(* CODESYS project GVL_CELL_MANAGER.gvl.xml

Project tree, tasks and I/O mapping:
  global variables GVL_CELL_MANAGER
*)

// GVL_CELL_MANAGER
{attribute 'qualified_only'}
VAR_GLOBAL
	Command : ST_CELL_COMMAND; // Команды менеджера ячейки
	Status  : ST_CELL_STATUS; // Рабочие статусы ячейки
	Diag    : ST_CELL_DIAG; // Состояние автомата ячейки
	Error   : ST_CELL_ERRORS; // Ошибки менеджера ячейки
END_VAR
